(* IEC 61131-3 sources: codesys-mcp-toolkit/standalone-sync/sources_st/511_05/Operations, 2 files *)

(* ---- FB_AutoCouplingDrainCascade.fb.st ---- *)
// @OBJECT_ID: 2cd08e36-15c9-47b1-a80c-451eef93a439
// @DECLARATION
FUNCTION_BLOCK FB_AutoCouplingDrainCascade
VAR_INPUT
    xStart             : BOOL;   // Триггер запуска стадии

    // --- Параметры Диазосоединения ---
    rFlowDiazoActual   : REAL;   // Текущий мгновенный расход диазо (м3/ч)
    rFlowDiazoSetpoint : REAL;   // Заданный мгновенный расход диазо

    // --- Параметры pH ---
    rPhActual          : REAL;   // Текущий pH (9.5..12 ед.)
    rPhSetpoint        : REAL;   // Уставка поддерживаемого pH

    // --- Условия завершения (Опустошение) ---
    rZeroFlowThreshold : REAL := 0.2;   // Порог "отсутствия расхода" (< 0.2 м3/ч)
    tEmptyDelay        : TIME := T#20S; // Время подтверждения отсутствия расхода

    // --- Настройки ПИД ---
    rKp_Diazo          : REAL := 1.0;
    rTn_Diazo          : REAL := 5.0;
    rTv_Diazo          : REAL := 0.0;
    rKp_pH             : REAL := 2.0;
    rTn_pH             : REAL := 10.0;
    rTv_pH             : REAL := 0.0;
END_VAR

VAR_IN_OUT
    rValveOutDiazo     : REAL;   // Задание на клапан диазо (0..100%)
    xAutoModeCmdDiazo  : BOOL;   // Режим АВТО для диазо
    rValveOutSoda      : REAL;   // Задание на клапан соды (0..100%)
    xAutoModeCmdSoda   : BOOL;   // Режим АВТО для соды
END_VAR

VAR_OUTPUT
    xActive            : BOOL;   // Стадия идет
    xDone              : BOOL;   // Стадия успешно завершена

    // --- Переменные для HMI ---
    rTimeLeft          : REAL;   // Оставшееся время до завершения (сек)
    rStateCode         : REAL;   // Код текущего состояния (0.0 .. 4.0)
    sStateStr          : STRING; // Текстовая расшифровка состояния
END_VAR

VAR
    fbPidFlowDiazo     : oscat_basic.CTRL_PID;
    fbPidPh            : oscat_basic.CTRL_PID;
    tonEmptyTimer      : TON;

    iState             : INT := 0; // Внутренний регистр шага State Machine
    xOldStart          : BOOL;
    xNeedStop          : BOOL;   // Флаг однократного останова оборудования
END_VAR

// @IMPLEMENTATION

// --- ЛОГИКА БЛОКА ---

// 1. Детектор старта (Исправление №1: Явный сброс выходов при старте)
IF xStart AND NOT xOldStart THEN
    iState     := 1;    // Переход в RUNNING
    xActive    := TRUE; // Явное включение
    xDone      := FALSE;// Явный сброс готовности
    xNeedStop  := FALSE;// Явный сброс команды останова

    xAutoModeCmdDiazo := TRUE;
    xAutoModeCmdSoda  := TRUE;
END_IF;

// 2. Детектор прерывания оператором
IF NOT xStart AND xOldStart AND (iState = 1 OR iState = 2) THEN
    iState := 4; // Переход в ABORTED
    xNeedStop := TRUE;
END_IF;

// 3. Вызов таймера опустошения
// Таймер работает ТОЛЬКО когда мы находимся на шаге 2 (EMPTYING)
tonEmptyTimer(
    IN := (iState = 2),
    PT := tEmptyDelay
);

// 4. КОНЕЧНЫЙ АВТОМАТ (STATE MACHINE)
CASE iState OF
    0: // --- IDLE (Ожидание) ---
        sStateStr  := 'ОЖИДАНИЕ: Аппарат готов к запуску';
        rStateCode := 0.0;
        xActive    := FALSE;
        xDone      := FALSE;
        rTimeLeft  := TIME_TO_REAL(tEmptyDelay) / 1000.0;

    1: // --- RUNNING (Нормальное регулирование) ---
        sStateStr  := 'РАБОТА: Поддержание расхода и pH';
        rStateCode := 1.0;
        xActive    := TRUE;
        xDone      := FALSE;
        rTimeLeft  := TIME_TO_REAL(tEmptyDelay) / 1000.0;

        // Условие перехода: расход упал ниже порога
        IF rFlowDiazoActual <= rZeroFlowThreshold THEN
            iState := 2;
        END_IF;

    2: // --- EMPTYING (Фиксация отсутствия расхода) ---
        sStateStr  := 'ВНИМАНИЕ: Падение расхода, отсчет времени...';
        rStateCode := 2.0;
        xActive    := TRUE;

        // Исправление №2: Безопасное вычитание времени (защита от переполнения/отрицательного результата)
        IF tonEmptyTimer.ET < tEmptyDelay THEN
            rTimeLeft := TIME_TO_REAL(tEmptyDelay - tonEmptyTimer.ET) / 1000.0;
        ELSE
            rTimeLeft := 0.0;
        END_IF;

        // Возврат в работу: если расход "ожил" (насос снова захватил жидкость)
        IF rFlowDiazoActual > rZeroFlowThreshold THEN
            iState := 1;

        // Успешное завершение: таймер досчитал до конца
        ELSIF tonEmptyTimer.Q THEN
            iState := 3;
            xNeedStop := TRUE; // Даем команду на закрытие клапанов
        END_IF;

    3: // --- DONE (Успешное завершение) ---
        sStateStr  := 'ЗАВЕРШЕНО: Емкость диазосоединения пуста';
        rStateCode := 3.0;
        xActive    := FALSE;
        xDone      := TRUE;
        rTimeLeft  := 0.0;

        // Исправление №3: Защита от гонки состояний при быстром повторном старте
        IF NOT xStart AND NOT xOldStart THEN
            iState := 0;
        END_IF;

    4: // --- ABORTED (Прервано оператором) ---
        sStateStr  := 'ПРЕРВАНО: Остановка по команде оператора';
        rStateCode := 4.0;
        xActive    := FALSE;
        xDone      := FALSE;
        rTimeLeft  := 0.0;

        // Исправление №3: Защита от гонки состояний при быстром повторном старте
        IF NOT xStart AND NOT xOldStart THEN
            iState := 0;
        END_IF;

END_CASE;

// 5. Вызов ПИД-регуляторов (Работают только на активных шагах 1 и 2)
IF iState = 1 OR iState = 2 THEN
    fbPidFlowDiazo(
        ACT := rFlowDiazoActual, SET := rFlowDiazoSetpoint,
        MAN := FALSE, RST := FALSE, KP := rKp_Diazo, TN := MAX(rTn_Diazo, 1.0),
        TV := rTv_Diazo, LL := 0.0, LH := 100.0
    );
    rValveOutDiazo := fbPidFlowDiazo.Y;

    fbPidPh(
        ACT := rPhActual, SET := rPhSetpoint,
        MAN := FALSE, RST := FALSE, KP := rKp_pH, TN := MAX(rTn_pH, 1.0),
        TV := rTv_pH, LL := 0.0, LH := 100.0
    );
    rValveOutSoda := fbPidPh.Y;
END_IF;

// 6. Однократный безопасный останов
IF xNeedStop THEN
    // Сбрасываем интеграторы ПИД
    fbPidFlowDiazo(MAN := TRUE, SET := 0.0, ACT := 0.0, RST := TRUE);
    fbPidPh(MAN := TRUE, SET := 0.0, ACT := 0.0, RST := TRUE);

    // Закрываем клапаны и возвращаем в ручной режим
    rValveOutDiazo    := 0.0;
    xAutoModeCmdDiazo := FALSE;
    rValveOutSoda     := 0.0;
    xAutoModeCmdSoda  := FALSE;

    xNeedStop := FALSE; // Сбрасываем триггер останова
END_IF;

xOldStart := xStart;

(* ---- FB_WaterLoading.fb.st ---- *)
// @OBJECT_ID: 8982d891-ac0a-4f55-8094-276c0250f702
// @DECLARATION
(*
    ФУНКЦИОНАЛЬНЫЙ БЛОК: FB_WaterLoading
    ВЕРСИЯ: 2.0.0
    ОПИСАНИЕ: Автоматическая загрузка воды заданной дозой.

    ЛОГИКА:
      - xStart OFF→ON  : старт → открываем клапан (xAutoControl:=TRUE), фиксируем объём
      - xStart ON→OFF  : прерывание оператором → закрываем клапан (xAutoControl:=FALSE)
      - Доза выполнена : rLoaded >= rDose - rDeadband → закрываем клапан, xStart:=FALSE

    ВАЖНО: xMode и xAutoControl — VAR_IN_OUT (прямая ссылка на внешние переменные).
           Присвоение только по триггеру (фронт старта, фронт стопа, завершение дозы).
           В рабочем цикле (xRunning=TRUE) — только обновление rLoaded, клапан не трогаем.

    СТАТУСЫ (rStatus):
      0.0 = IDLE
      1.0 = RUNNING
      2.0 = DONE
      3.0 = ABORTED
*)
 (*
    ФУНКЦИОНАЛЬНЫЙ БЛОК: FB_WaterLoading
    ВЕРСИЯ: 2.1.0 (Исправленная)
*)

FUNCTION_BLOCK FB_WaterLoading
VAR_INPUT
    rTotalVolume    : REAL;   (* Текущий объём сумматора расходомера, куб.м *)
    rDose           : REAL;   (* Заданная доза, куб.м *)
    rDeadband       : REAL;   (* Мёртвый остаток для предиктивного закрытия, куб.м *)
END_VAR
VAR_IN_OUT
    xStart          : BOOL;   (* Команда: ON=старт, OFF=стоп/прерывание *)
    xMode           : BOOL;   (* Режим клапана: FALSE=ручной, TRUE=авто *)
    xAutoControl    : BOOL;   (* Автозадание клапана *)
END_VAR
VAR_OUTPUT
    rLoaded         : REAL;   (* Загружено в текущем цикле, куб.м *)
    rStatus         : REAL;   (* 0=IDLE 1=RUNNING 2=DONE 3=ABORTED *)
END_VAR
VAR
    rStartVolume    : REAL;
    xLastStart      : BOOL;
    xRunning        : BOOL;
END_VAR

// @IMPLEMENTATION
// ----------------------------------------------------------------
// ФРОНТ OFF→ON : СТАРТ ДОЗИРОВАНИЯ
// ----------------------------------------------------------------
IF xStart AND NOT xLastStart THEN
    rStartVolume := rTotalVolume;
    rLoaded      := 0.0;
    xRunning     := TRUE;
    rStatus      := 1.0;
    xMode        := TRUE;   // переключаем клапан в авторежим
    xAutoControl := TRUE;   // открываем клапан
END_IF;

// ----------------------------------------------------------------
// РАБОЧИЙ ЦИКЛ: Считаем объем и проверяем достижение дозы
// ----------------------------------------------------------------
IF xRunning THEN
    rLoaded := rTotalVolume - rStartVolume;

    // Доза выполнена — предиктивное закрытие (Высший приоритет)
    IF rLoaded >= (rDose - rDeadband) THEN
        xAutoControl := FALSE;  // закрываем клапан
        xRunning     := FALSE;
        xStart       := FALSE;  // автосброс команды
        rStatus      := 2.0;    // DONE
    END_IF;
END_IF;

// ----------------------------------------------------------------
// ФРОНТ ON→OFF : ПРЕРЫВАНИЕ ОПЕРАТОРОМ
// (Сработает только если доза ЕЩЕ НЕ выполнена в этом цикле)
// ----------------------------------------------------------------
IF NOT xStart AND xLastStart AND xRunning THEN
    xRunning     := FALSE;
    xAutoControl := FALSE;  // закрываем клапан
    rStatus      := 3.0;    // ABORTED
END_IF;

// ----------------------------------------------------------------
// БУФЕР ФРОНТА (в конце скана)
// ----------------------------------------------------------------
xLastStart := xStart;
